FUNCTION F_UpdateEvent
VAR_INPUT
	stEvent				: REFERENCE TO ST_Event;
END_VAR
VAR
	fbGETSYSTEMTIME 	: GETSYSTEMTIME;
	stFileTime 			: T_FILETIME;
END_VAR

fbGETSYSTEMTIME(timeLoDW=> stFileTime.dwLowDateTime, 
				timeHiDW=> stFileTime.dwHighDateTime);
stEvent.dtTimeStamp:= FILETIME_TO_DT(fileTime:=stFileTime);

END_FUNCTION

(* stored: Version 1.1.0.1, ProductVersion 3.1.4024.12
   POU F_UpdateEvent: Id {e8bdd8de-7c16-42be-8873-53eba818ece5}, SpecialFunc None *)
